INTERFACE I_ContentAddedEvent EXTENDS I_Event

PROPERTY PUBLIC Target : I_Content
GET
END_GET
END_PROPERTY

END_INTERFACE

(* stored: Version 1.1.0.1, ProductVersion 3.1.4024.12
   Itf I_ContentAddedEvent: Id {90739cbb-767e-049e-1d6c-6f8bb5e021b5}
   Property Target: Id {1be8ae1a-e31a-00e0-3123-40f0b64730c9}
   Get Get: Id {c7273ec6-7e0e-00c7-1683-9b4fba0d89c0} *)
